TYPE ST_EtherCATState :
STRUCT
	EtherCATState : BOOL;
	CRCPortA :UDINT;
	CRCPortB :UDINT;
	CRCPortC :UDINT;
END_STRUCT
END_TYPE

(* stored: Version 1.1.0.1, ProductVersion 3.1.4024.12
   DUT ST_EtherCATState: Id {9837df17-f8ca-4b15-9565-f594c53cf714} *)
